(* CODESYS project Fluke.library
   Company: Ziga Javornik
   DefaultNamespace: ZigaLibs.Fluke
   Version: 0.0.1.0
   Placeholder: ZigaLibs.Fluke
   Author: Ziga Javornik
   Title: ZigaLibs.Fluke

Project tree, tasks and I/O mapping:
  libraries: Tc2_Standard, * (Beckhoff Automation GmbH); Tc2_System, * (Beckhoff Automation GmbH); Tc3_Module, * (Beckhoff Automation GmbH); TcUnit, 1.3.1 (www.tcunit.org); ZigaLibs.Core, 0.0.3.7 (Ziga Javornik); ZigaLibs.Logging, 0.0.4.1 (Ziga Javornik); ZigaLibs.TcpIp, 0.0.2.2 (Ziga Javornik)
  GVLs/
  SOURCE/
    Endurance IR Pyrometers/
      DUTs/
        data type ST_EndurancePyrometerCommands
        data type ST_EndurancePyrometerCommParameters
        data type ST_EndurancePyrometerErrorCodes
        data type ST_EndurancePyrometerErrorResponse
      GVLs/
        global variables GVL_Params_EndurancePyrometer
      POUs/
        program EndurancePyrometerConstants [ST]
        function block FB_EndurancePyrometer [ST]: FB_init, CreateSendCommand, ExtractResponse, GetLogPrefix, LogError, LogInfo, LogWarning, RemoveResponsePrefix, RemoveResponseSuffix, ValidateLogger, CommParameters
  TESTS/
    Test suites/
      function block FB_EndurancePyrometer_Tests [ST]: Test00_AttenuationTooHigh_ExpectMaxTemp, Test01_HeaterTemperatureOverrange_ExpectMaxTemp, Test02_HeaterTemperatureUnderrange_ExpectMaxTemp, Test03_InternalTemperatureTooHigh_ExpectMaxTemp, Test04_InternalTemperatureTooLow_ExpectMaxTemp, Test05_SyntaxError_ExpectMaxTemp, Test06_TemperatureOverrange_ExpectMaxTemp, Test07_TemperatureUnderrange_ExpectMinTemp
      function block FB_EndurancePyrometerConstants_Tests [ST]: Test01_ErrorCodesValues
    program PRG_TESTS [ST]
*)

// SOURCE/Endurance IR Pyrometers/DUTs/ST_EndurancePyrometerCommands
TYPE ST_EndurancePyrometerCommands :
STRUCT
	ReadTemperatureCommand 			: STRING := '?T';	// Asks the pyrometer for current temperature
	ReadSensorInternalTemperature	: STRING := '?I';	// Asks for the internal temperature of the sensor
	ReadTargetTemperatureEnergy		: STRING := '?Q';	// Asks for the energy value of the target temperature
	ReadEmissivity					: STRING := '?E';	// Asks for the current emissivity value
	SetEmissivity					: STRING := 'E=';	// Command for setting emissivity, followed value will be set
	SetTemperatuerPhysicalUnit_C	: STRING := 'U=C';	// Sets the physical unit for temperature to °C
	SetTemperatuerPhysicalUnit_F	: STRING := 'U=F';	// Sets the physical unit for temperature to °F
	
	ResponseSuffix			: STRING := '$R$N';	// Response from pyrometer ends with the suffix
	ResponsePrefix			: STRING := '!';	// Response from pyrometer starts with the prefix
	CommandSuffix 			: STRING := '$R';	// Every command needs to end with the suffix
END_STRUCT
END_TYPE

// SOURCE/Endurance IR Pyrometers/DUTs/ST_EndurancePyrometerCommParameters
TYPE ST_EndurancePyrometerCommParameters :
STRUCT
	ReadCycle		: TIME := T#500MS;	// Cyclic reading of certain values is executed within the interval defined by this parameter.
	ReconnectPeriod	: TIME := T#45S;	// Reconnect period for TCP/IP. Don't set too low (30s should be the lowest)
	Ipv4Address		: Tc2_System.T_IPv4Addr := '192.168.42.132';	// IPV4 address of the device.
	Port			: ZigaLibs_TcpIp.T_Port := 6363;	// Port of the device.
END_STRUCT
END_TYPE

// SOURCE/Endurance IR Pyrometers/DUTs/ST_EndurancePyrometerErrorCodes
(*When an error or failure does occur, the temperature display indicates the possible failure area and the output
circuits automatically adjust to the lowest or highest preset level. The following table shows the corresponding
values and the error code transmitted over the digital interface.

Fail safe error codes, from: https://media.fluke.com/048723ef-592e-4cbc-86d4-b4ad00bf9a87_original%20file.pdf

Condition 											2-color 			1-color(wide band)**	1-color*(narrow band)**
Heater temperature over range, >= 80°C (176°F) 		ECHH 				ECHH 					ECHH
Heater temperature under range, <= 50°C (122°F) 	ECUU 				ECUU 					ECUU
Internal temperature over range, >= 85°C (185°F) 	EIHH 				EIHH 					EIHH
Internal temperature under range, <= 0°C (32°F) 	EIUU 				EIUU 					EIUU
Wide band detector failure 							EHHH	 			EHHH 					<temperature>
Narrow band detector failure 						EHHH 				<temperature> 			EHHH
Energy too low 										EUUU 				<temperature> 			<temperature>
Attenuation too high (>95%)*** 						EAAA 				<temperature> 			<temperature>
Attenuation too high >95%
("dirty lens", relay will go to “alarm” state)***	<temperature> 		<temperature> 			<temperature>
2-color temperature under range 					EUUU 				<temperature> 			<temperature>
2-color temperature over range 						EHHH 				<temperature> 			<temperature>
Wide band temperature under range 					<temperature> 		EUUU 					<temperature>
Wide band temperature over range 					<temperature> 		EHHH 					<temperature>
Narrow band temperature under range 				<temperature> 		<temperature> 			EUUU
Narrow band temperature over range 					<temperature> 		<temperature> 			EHHH


* only available via ASCII command
** wide and narrow band stands for the first and the second wavelength in 2-color mode
*** note that the activation levels for these conditions may be set to different values (e.g., "dirty lens" at 95%, EAAA at 98%)
*)
TYPE ST_EndurancePyrometerErrorCodes :
STRUCT
	TemperatureOverrange		: ST_EndurancePyrometerErrorResponse := (Code := 'EHHH', Message := 'Temperature over  range');
	TemperatureUnderrange		: ST_EndurancePyrometerErrorResponse := (Code := 'EUUU', Message := 'Temperature under range');
	InternalTemperatureTooLow	: ST_EndurancePyrometerErrorResponse := (Code := 'EIUU', Message := 'Internal temperature under range, <= 0°C (32°F) ');
	InternalTemperatureTooHigh	: ST_EndurancePyrometerErrorResponse := (Code := 'EIHH', Message := 'Internal temperature over range, >= 85°C (185°F)');
	AttenuationTooHigh			: ST_EndurancePyrometerErrorResponse := (Code := 'EAAA', Message := 'Attenuation too high (>95%)');
	HeaterTemperatureUnderrange	: ST_EndurancePyrometerErrorResponse := (Code := 'ECUU', Message := 'Heater temperature under range, <= 50°C (122°F) ');
	HeaterTemperatureOverrange	: ST_EndurancePyrometerErrorResponse := (Code := 'ECHH', Message := 'Heater temperature over range, >= 80°C (176°F)');
	SyntaxError					: ST_EndurancePyrometerErrorResponse := (Code := '*Syntax Error', Message := 'A value entered in an incorrect format');
END_STRUCT
END_TYPE

// SOURCE/Endurance IR Pyrometers/DUTs/ST_EndurancePyrometerErrorResponse
TYPE ST_EndurancePyrometerErrorResponse :
STRUCT
	Code	: Tc2_System.T_MaxString;
	Message	: STRING;
END_STRUCT
END_TYPE

// SOURCE/Endurance IR Pyrometers/GVLs/GVL_Params_EndurancePyrometer
{attribute 'qualified_only'}
VAR_GLOBAL CONSTANT
	MAX_TEMPERATURE	: REAL := 3000.0;	// Sets the maximum temperature of the pyromerer - should be set accordingly to pyrometer series
	MIN_TEMPERATURE	: REAL := 1000.0;	// Sets the minimum temperatuer of the pyrometer - should be set accordingly to pyrometer series
END_VAR

// SOURCE/Endurance IR Pyrometers/POUs/EndurancePyrometerConstants
PROGRAM EndurancePyrometerConstants
VAR CONSTANT
	ErrorCodes	: ST_EndurancePyrometerErrorCodes;
	Commands	: ST_EndurancePyrometerCommands;	
END_VAR

END_PROGRAM

// SOURCE/Endurance IR Pyrometers/POUs/FB_EndurancePyrometer
FUNCTION_BLOCK FB_EndurancePyrometer EXTENDS ZigaLibs_Core.FB_HasInstanceNameAndPath
VAR_INPUT
	connect		: BOOL;
	readCycle	: TIME;	// Read cycle, should not be set under 300ms, limitation is done within
	ipAddress	: Tc2_System.T_IPv4Addr;
	port		: UINT;	
END_VAR

VAR_OUTPUT
	temperature	: REAL;
	error		: BOOL;
	connected	: BOOL;
	errorCode	: Tc2_System.T_MaxString;
END_VAR

VAR
	_tcpIp			: ZigaLibs_TcpIp.FB_TcpIpCommControl(_logger);
	_reconnectTimer	: Tc2_Standard.TON;
	_readTimer		: Tc2_Standard.TON;
	_readWriteStep	:(READY, SEND_READ_COMMAND, AWAIT_RESPONSE);
	_response		: Tc2_System.T_MaxString;
	_logger			: REFERENCE TO ZigaLibs_Logging.I_Logger;
	_commParameters	: ST_EndurancePyrometerCommParameters;
	_readTemperatureCommand	: STRING;	
	_sb				: ZigaLibs_Core.FB_StringBuilder;
END_VAR

_tcpIp.ReconnectPeriod := T#10S;

_reconnectTimer(
	IN := NOT _reconnectTimer.Q AND _tcpIp.Error, 
	PT := T#30S);

// Communication via TcpIp
IF connect THEN
	IF _reconnectTimer.Q THEN
		_tcpIp.Disconnect();
	ELSIF NOT _tcpIp.IsConnected THEN
		_tcpIp.Connect(ipAddress, port);		
	END_IF
ELSE
	_tcpIp.Disconnect();
END_IF

connected := _tcpIp.IsConnected;
_tcpIp();

IF _tcpIp.IsConnected THEN
	_readTimer(PT := MIN (T#200MS, readCycle));
	
	CASE _readWriteStep OF
		READY:
			_readTimer.IN := TRUE;
			IF _readTimer.Q THEN
				_readTimer.IN := FALSE;
				_readWriteStep := SEND_READ_COMMAND;
			END_IF
		
		SEND_READ_COMMAND:
			_readTemperatureCommand := CreateSendCommand(EndurancePyrometerConstants.Commands.ReadTemperatureCommand);
			IF _tcpIp.Send(_readTemperatureCommand) THEN
				_readWriteStep := AWAIT_RESPONSE;
			END_IF
		
		AWAIT_RESPONSE:
			IF _tcpIp.Receive(_response) THEN
				ExtractResponse('T');
				_readWriteStep := READY;
			END_IF
	END_CASE
ELSE
	// Tcp error - set temperature to max to prevent PID overheating.
	temperature := GVL_Params_EndurancePyrometer.MAX_TEMPERATURE;
END_IF

error := _tcpIp.Error OR error;

METHOD FB_init : BOOL
VAR_INPUT
	bInitRetains : BOOL; // if TRUE, the retain variables are initialized (warm start / cold start)
	bInCopyCode : BOOL;  // if TRUE, the instance afterwards gets moved into the copy code (online change)
	logger	: REFERENCE TO ZigaLibs_Logging.I_Logger;
END_VAR
_logger REF= logger;
END_METHOD

METHOD CreateSendCommand : STRING
VAR_INPUT
	command	: STRING;
END_VAR
CreateSendCommand := Tc2_Standard.CONCAT(command, EndurancePyrometerConstants.Commands.CommandSuffix);
END_METHOD

METHOD INTERNAL ExtractResponse
VAR_INPUT
	sentCommand	: STRING;
END_VAR

VAR
	response			: Tc2_System.T_MaxString;
	responseTmp			: Tc2_System.T_MaxString;
	suffixLength		: INT;

	suffixRemoveAttempt	: DINT;
END_VAR

VAR_INST
	syntaxErrorTrigger	: Tc2_Standard.R_TRIG;
	errorTrigger		: Tc2_Standard.R_TRIG;
	errorClearedTrigge	: Tc2_Standard.F_TRIG;
	sb					: ZigaLibs_Core.FB_StringBuilder;
END_VAR
response := _response;
syntaxErrorTrigger();

// Syntax error - return early
IF Tc2_Standard.FIND(response, EndurancePyrometerConstants.ErrorCodes.SyntaxError.Code) <> 0 THEN
	syntaxErrorTrigger(CLK := TRUE);
	IF syntaxErrorTrigger.Q THEN
		LogError(_sb.Reset()
			.AddString('Syntax error! Sent command is ')
			.AddWithDblQuotationMarks(sentCommand)
			.AddString('.')
			.Create());
	END_IF
	error := TRUE;
	errorCode := 'Syntax error';
	temperature := GVL_Params_EndurancePyrometer.MAX_TEMPERATURE;
	RETURN;
END_IF

syntaxErrorTrigger.CLK := FALSE;

response := RemoveResponsePrefix(sentCommand, response);	
response := RemoveResponseSuffix(response);

error := FALSE;

// Parse response
IF response = EndurancePyrometerConstants.ErrorCodes.TemperatureOverrange.Code THEN
	errorCode := EndurancePyrometerConstants.ErrorCodes.TemperatureOverrange.Message;
	temperature := GVL_Params_EndurancePyrometer.MAX_TEMPERATURE;
ELSIF response = EndurancePyrometerConstants.ErrorCodes.TemperatureUnderrange.Code THEN
	errorCode := EndurancePyrometerConstants.ErrorCodes.TemperatureUnderrange.Message;	
	temperature := GVL_Params_EndurancePyrometer.MIN_TEMPERATURE;	
ELSIF response = EndurancePyrometerConstants.ErrorCodes.InternalTemperatureTooLow.Code THEN
	errorCode := EndurancePyrometerConstants.ErrorCodes.InternalTemperatureTooLow.Message;
	temperature := GVL_Params_EndurancePyrometer.MAX_TEMPERATURE;
	error := TRUE;	
ELSIF response = EndurancePyrometerConstants.ErrorCodes.InternalTemperatureTooHigh.Code THEN
	errorCode := EndurancePyrometerConstants.ErrorCodes.InternalTemperatureTooHigh.Message;
	temperature := GVL_Params_EndurancePyrometer.MAX_TEMPERATURE;
	error := TRUE;	
ELSIF response = EndurancePyrometerConstants.ErrorCodes.AttenuationTooHigh.Code THEN
	errorCode := EndurancePyrometerConstants.ErrorCodes.AttenuationTooHigh.Message;
	temperature := GVL_Params_EndurancePyrometer.MAX_TEMPERATURE;
	error := TRUE;	
ELSIF response = EndurancePyrometerConstants.ErrorCodes.HeaterTemperatureUnderrange.Code THEN
	errorCode := EndurancePyrometerConstants.ErrorCodes.HeaterTemperatureUnderrange.Message;
	temperature := GVL_Params_EndurancePyrometer.MAX_TEMPERATURE;
	error := TRUE;	
ELSIF response = EndurancePyrometerConstants.ErrorCodes.HeaterTemperatureOverrange.Code THEN
	errorCode := EndurancePyrometerConstants.ErrorCodes.HeaterTemperatureOverrange.Message;
	temperature := GVL_Params_EndurancePyrometer.MAX_TEMPERATURE;
	error := TRUE;	
ELSE	
	errorCode := 'No error';
	temperature := STRING_TO_REAL(response);	
END_IF

errorTrigger(CLK := errorCode <> 'No error');
IF errorTrigger.Q THEN
	IF __ISVALIDREF(_logger) THEN
		_logger.LogError(_sb.Reset()
			.AddString(GetLogPrefix())
			.AddString('Pyrometer response indicates error! Error description: ')
			.AddWithDblQuotationMarks(errorCode)
			.AddString('.')
			.Create());
	END_IF	
END_IF

errorClearedTrigge(CLK := errorCode = 'No error');
IF errorClearedTrigge.Q THEN
	IF __ISVALIDREF(_logger) THEN
		_logger.LogInfo(_sb.Reset()
			.AddString(GetLogPrefix())
			.AddString('Previous pyrometer error code is no longer active.')
			.Create());
	END_IF	
END_IF
END_METHOD

METHOD PROTECTED GetLogPrefix : T_MaxString
VAR_INPUT
END_VAR

VAR
	sb	: ZigaLibs_Core.FB_StringBuilder;
END_VAR
GetLogPrefix := sb.AddString(THIS^.InstanceName)
	.AddString(' ')
	.AddWithDblQuotationMarks(ipAddress)
	.AddString(': ')
	.Create();
END_METHOD

METHOD PROTECTED LogError
VAR_INPUT
	message	: Tc2_System.T_MaxString;
END_VAR 
VAR
	sb	: ZigaLibs_Core.FB_StringBuilder;
END_VAR
IF NOT ValidateLogger() THEN
	RETURN;
END_IF

_logger.LogError(
	sb.AddString(GetLogPrefix())
		.AddString(message)
		.Create());
END_METHOD

METHOD PROTECTED LogInfo
VAR_INPUT
	message	: Tc2_System.T_MaxString;
END_VAR 
VAR
	sb	: ZigaLibs_Core.FB_StringBuilder;
END_VAR
IF NOT ValidateLogger() THEN
	RETURN;
END_IF

_logger.LogInfo(
	sb.AddString(GetLogPrefix())
		.AddString(message)
		.Create());
END_METHOD

METHOD PROTECTED LogWarning
VAR_INPUT
	message : Tc2_System.T_MaxString;
END_VAR
VAR
	sb	: ZigaLibs_Core.FB_StringBuilder;
END_VAR
IF NOT ValidateLogger() THEN
	RETURN;
END_IF

_logger.LogWarning(
	sb.AddString(GetLogPrefix())
		.AddString(message)
		.Create());
END_METHOD

// Removes the prefix from the received response and returns the trimmer string
METHOD PROTECTED RemoveResponsePrefix : Tc2_System.T_MaxString
VAR_INPUT
	sentCommand	: Tc2_System.T_MaxString;
	response	: Tc2_System.T_MaxString;
END_VAR
// Remove prefix
RemoveResponsePrefix := Tc2_Standard.DELETE(
	STR := response, 
	LEN := Tc2_Standard.LEN(sentCommand) + LEN(EndurancePyrometerConstants.Commands.ResponsePrefix),
	POS := 1);
END_METHOD

// Removes the suffix from the received response and returns the trimmer string
METHOD PROTECTED RemoveResponseSuffix : T_MaxString
VAR_INPUT
	response	: STRING;
END_VAR
VAR
	suffixPosition	: INT;	
	trimmedResponse		: STRING;
END_VAR

// Remove suffix - sometimes the suffix is sent in multiples (no idea why Fluke does this), remove all occurences!	
suffixPosition := Tc2_Standard.FIND(STR1 := response, STR2 := EndurancePyrometerConstants.Commands.ResponseSuffix);
trimmedResponse := response;
IF suffixPosition <> 0 THEN
	response := Tc2_Standard.LEFT(STR := trimmedResponse, SIZE := suffixPosition - 1);		
END_IF

RemoveResponseSuffix := trimmedResponse;
END_METHOD

METHOD PROTECTED ValidateLogger : BOOL
VAR_INPUT
END_VAR
ValidateLogger := __ISVALIDREF(_logger);
END_METHOD

// Gets or sets communication parameters of the device.
PROPERTY PUBLIC CommParameters : REFERENCE TO ST_EndurancePyrometerCommParameters
GET
CommParameters REF= _commParameters;
END_GET
SET
_commParameters := CommParameters;
END_SET
END_PROPERTY

END_FUNCTION_BLOCK

// TESTS/Test suites/FB_EndurancePyrometer_Tests
// Subject under test
FUNCTION_BLOCK INTERNAL FB_EndurancePyrometer_Tests EXTENDS FB_TestSuite

// Create instance variables that will be accesible for all tests
VAR
END_VAR

// Call your test methods here
Test00_AttenuationTooHigh_ExpectMaxTemp();
Test01_HeaterTemperatureOverrange_ExpectMaxTemp();
Test02_HeaterTemperatureUnderrange_ExpectMaxTemp();
Test03_InternalTemperatureTooHigh_ExpectMaxTemp();
Test04_InternalTemperatureTooLow_ExpectMaxTemp();
Test05_SyntaxError_ExpectMaxTemp();
Test06_TemperatureOverrange_ExpectMaxTemp();
Test07_TemperatureUnderrange_ExpectMinTemp();

METHOD PRIVATE Test00_AttenuationTooHigh_ExpectMaxTemp

(* Instanced variables are VERY useful for writing tests since tests are run in paralel (by default).
By instantiating local variables that are not placed on the same stack as method (values are retained between calls)
you make sure that the SUT is not changed by some other test. *)
VAR_INST
	
END_VAR

// Place temporary variables here
VAR
	pyrometer	: FB_EndurancePyrometer(0);
END_VAR
// The name of the test, is the same as method name!
// Use this for paralel unit tests
// TcUnit.TEST('TestXX_Template');

// Use this for running tests in sequence
IF TcUnit.TEST_ORDERED('Test00_AttenuationTooHigh_ExpectMaxTemp') THEN
	
	TcUnit.WRITE_PROTECTED_STRING(
		ADR(pyrometer._response), 
		CONCAT('!T', EndurancePyrometerConstants.ErrorCodes.AttenuationTooHigh.Code));
		
	pyrometer.ExtractResponse('T');
	AssertEquals_REAL(
		Actual := pyrometer.temperature,
		Expected := GVL_Params_EndurancePyrometer.MAX_TEMPERATURE,
		Delta := 0.1,
		Message := '');
		
	AssertTrue(Condition := pyrometer.error, Message := 'Attenuation too high should trigger an error');
	TcUnit.TEST_FINISHED();	
END_IF
END_METHOD

METHOD PRIVATE Test01_HeaterTemperatureOverrange_ExpectMaxTemp

(* Instanced variables are VERY useful for writing tests since tests are run in paralel (by default).
By instantiating local variables that are not placed on the same stack as method (values are retained between calls)
you make sure that the SUT is not changed by some other test. *)
VAR_INST
	
END_VAR

// Place temporary variables here
VAR
	pyrometer	: FB_EndurancePyrometer(0);
END_VAR
// The name of the test, is the same as method name!
// Use this for paralel unit tests
// TcUnit.TEST('TestXX_Template');

// Use this for running tests in sequence
IF TcUnit.TEST_ORDERED('Test01_HeaterTemperatureOverrange_ExpectMaxTemp') THEN
	
	TcUnit.WRITE_PROTECTED_STRING(
		ADR(pyrometer._response), 
		CONCAT('!T', EndurancePyrometerConstants.ErrorCodes.HeaterTemperatureOverrange.Code));
		
	pyrometer.ExtractResponse('T');
	AssertEquals_REAL(
		Actual := pyrometer.temperature,
		Expected := GVL_Params_EndurancePyrometer.MAX_TEMPERATURE,
		Delta := 0.1,
		Message := '');

	AssertTrue(Condition := pyrometer.error, Message := 'Heater temperature overrange should trigger an error');
	TcUnit.TEST_FINISHED();	
END_IF
END_METHOD

METHOD PRIVATE Test02_HeaterTemperatureUnderrange_ExpectMaxTemp

(* Instanced variables are VERY useful for writing tests since tests are run in paralel (by default).
By instantiating local variables that are not placed on the same stack as method (values are retained between calls)
you make sure that the SUT is not changed by some other test. *)
VAR_INST
	
END_VAR

// Place temporary variables here
VAR
	pyrometer	: FB_EndurancePyrometer(0);
END_VAR
// The name of the test, is the same as method name!
// Use this for paralel unit tests
// TcUnit.TEST('TestXX_Template');

// Use this for running tests in sequence
IF TcUnit.TEST_ORDERED('Test02_HeaterTemperatureUnderrange_ExpectMaxTemp') THEN
	
	TcUnit.WRITE_PROTECTED_STRING(
		ADR(pyrometer._response), 
		CONCAT('!T', EndurancePyrometerConstants.ErrorCodes.HeaterTemperatureUnderrange.Code));
		
	pyrometer.ExtractResponse('T');
	AssertEquals_REAL(
		Actual := pyrometer.temperature,
		Expected := GVL_Params_EndurancePyrometer.MAX_TEMPERATURE,
		Delta := 0.1,
		Message := '');
		
	AssertTrue(Condition := pyrometer.error, Message := ' Heater temperature underrange should trigger an error');		
	TcUnit.TEST_FINISHED();	
END_IF
END_METHOD

METHOD PRIVATE Test03_InternalTemperatureTooHigh_ExpectMaxTemp

(* Instanced variables are VERY useful for writing tests since tests are run in paralel (by default).
By instantiating local variables that are not placed on the same stack as method (values are retained between calls)
you make sure that the SUT is not changed by some other test. *)
VAR_INST
	
END_VAR

// Place temporary variables here
VAR
	pyrometer	: FB_EndurancePyrometer(0);
END_VAR
// The name of the test, is the same as method name!
// Use this for paralel unit tests
// TcUnit.TEST('TestXX_Template');

// Use this for running tests in sequence
IF TcUnit.TEST_ORDERED('Test03_InternalTemperatureTooHigh_ExpectMaxTemp') THEN
	
	TcUnit.WRITE_PROTECTED_STRING(
		ADR(pyrometer._response), 
		CONCAT('!T', EndurancePyrometerConstants.ErrorCodes.InternalTemperatureTooHigh.Code));
		
	pyrometer.ExtractResponse('T');
	AssertEquals_REAL(
		Actual := pyrometer.temperature,
		Expected := GVL_Params_EndurancePyrometer.MAX_TEMPERATURE,
		Delta := 0.1,
		Message := '');
		
	AssertTrue(Condition := pyrometer.error, Message := 'Internal temperature too high should trigger an error');	
	TcUnit.TEST_FINISHED();	
END_IF
END_METHOD

METHOD PRIVATE Test04_InternalTemperatureTooLow_ExpectMaxTemp

(* Instanced variables are VERY useful for writing tests since tests are run in paralel (by default).
By instantiating local variables that are not placed on the same stack as method (values are retained between calls)
you make sure that the SUT is not changed by some other test. *)
VAR_INST
	
END_VAR

// Place temporary variables here
VAR
	pyrometer	: FB_EndurancePyrometer(0);
END_VAR
// The name of the test, is the same as method name!
// Use this for paralel unit tests
// TcUnit.TEST('TestXX_Template');

// Use this for running tests in sequence
IF TcUnit.TEST_ORDERED('Test04_InternalTemperatureTooLow_ExpectMaxTemp') THEN
	
	TcUnit.WRITE_PROTECTED_STRING(
		ADR(pyrometer._response), 
		CONCAT('!T', EndurancePyrometerConstants.ErrorCodes.InternalTemperatureTooLow.Code));
		
	pyrometer.ExtractResponse('T');
	AssertEquals_REAL(
		Actual := pyrometer.temperature,
		Expected := GVL_Params_EndurancePyrometer.MAX_TEMPERATURE,
		Delta := 0.1,
		Message := '');
		
	AssertTrue(Condition := pyrometer.error, Message := 'Internal tempereature too low should trigger an error');	
	TcUnit.TEST_FINISHED();	
END_IF
END_METHOD

METHOD PRIVATE Test05_SyntaxError_ExpectMaxTemp

(* Instanced variables are VERY useful for writing tests since tests are run in paralel (by default).
By instantiating local variables that are not placed on the same stack as method (values are retained between calls)
you make sure that the SUT is not changed by some other test. *)
VAR_INST
	
END_VAR

// Place temporary variables here
VAR
	pyrometer	: FB_EndurancePyrometer(0);
END_VAR
// The name of the test, is the same as method name!
// Use this for paralel unit tests
// TcUnit.TEST('TestXX_Template');

// Use this for running tests in sequence
IF TcUnit.TEST_ORDERED('Test05_SyntaxError_ExpectMaxTemp') THEN
	
	TcUnit.WRITE_PROTECTED_STRING(
		ADR(pyrometer._response), 
		CONCAT('!T', EndurancePyrometerConstants.ErrorCodes.SyntaxError.Code));
		
	pyrometer.ExtractResponse('T');
	AssertEquals_REAL(
		Actual := pyrometer.temperature,
		Expected := GVL_Params_EndurancePyrometer.MAX_TEMPERATURE,
		Delta := 0.1,
		Message := '');
		
	AssertTrue(Condition := pyrometer.error, Message := 'Syntax error should trigger an error');	
	TcUnit.TEST_FINISHED();	
END_IF
END_METHOD

METHOD PRIVATE Test06_TemperatureOverrange_ExpectMaxTemp

(* Instanced variables are VERY useful for writing tests since tests are run in paralel (by default).
By instantiating local variables that are not placed on the same stack as method (values are retained between calls)
you make sure that the SUT is not changed by some other test. *)
VAR_INST
	
END_VAR

// Place temporary variables here
VAR
	pyrometer	: FB_EndurancePyrometer(0);
END_VAR
// The name of the test, is the same as method name!
// Use this for paralel unit tests
// TcUnit.TEST('TestXX_Template');

// Use this for running tests in sequence
IF TcUnit.TEST_ORDERED('Test06_TemperatureOverrange_ExpectMaxTemp') THEN
	
	TcUnit.WRITE_PROTECTED_STRING(
		ADR(pyrometer._response), 
		CONCAT('!T', EndurancePyrometerConstants.ErrorCodes.TemperatureOverrange.Code));
		
	pyrometer.ExtractResponse('T');
	AssertEquals_REAL(
		Actual := pyrometer.temperature,
		Expected := GVL_Params_EndurancePyrometer.MAX_TEMPERATURE,
		Delta := 0.1,
		Message := '');
		
	AssertFalse(Condition := pyrometer.error, Message := 'Temperature overrange should not trigger an error');	
	TcUnit.TEST_FINISHED();	
END_IF
END_METHOD

METHOD PRIVATE Test07_TemperatureUnderrange_ExpectMinTemp

(* Instanced variables are VERY useful for writing tests since tests are run in paralel (by default).
By instantiating local variables that are not placed on the same stack as method (values are retained between calls)
you make sure that the SUT is not changed by some other test. *)
VAR_INST
	
END_VAR

// Place temporary variables here
VAR
	pyrometer	: FB_EndurancePyrometer(0);
END_VAR
// The name of the test, is the same as method name!
// Use this for paralel unit tests
// TcUnit.TEST('TestXX_Template');

// Use this for running tests in sequence
IF TcUnit.TEST_ORDERED('Test07_TemperatureUnderrange_ExpectMinTemp') THEN
	
	TcUnit.WRITE_PROTECTED_STRING(
		ADR(pyrometer._response), 
		CONCAT('!T', EndurancePyrometerConstants.ErrorCodes.TemperatureUnderrange.Code));
		
	pyrometer.ExtractResponse('T');
	AssertEquals_REAL(
		Actual := pyrometer.temperature,
		Expected := GVL_Params_EndurancePyrometer.MIN_TEMPERATURE,
		Delta := 0.1,
		Message := '');
	
	AssertFalse(Condition := pyrometer.error, Message := 'Temperature underrange should not trigger an error');	
	TcUnit.TEST_FINISHED();	
END_IF
END_METHOD

END_FUNCTION_BLOCK

// TESTS/Test suites/FB_EndurancePyrometerConstants_Tests
FUNCTION_BLOCK INTERNAL FB_EndurancePyrometerConstants_Tests EXTENDS FB_TestSuite
VAR_INPUT
END_VAR
VAR_OUTPUT
END_VAR
VAR
END_VAR

Test01_ErrorCodesValues();

METHOD PRIVATE Test01_ErrorCodesValues
(*
Fail safe error codes, from: https://media.fluke.com/048723ef-592e-4cbc-86d4-b4ad00bf9a87_original%20file.pdf

Condition 											2-color 			1-color(wide band)**	1-color*(narrow band)**
Heater temperature over range, >= 80°C (176°F) 		ECHH 				ECHH 					ECHH
Heater temperature under range, <= 50°C (122°F) 	ECUU 				ECUU 					ECUU
Internal temperature over range, >= 85°C (185°F) 	EIHH 				EIHH 					EIHH
Internal temperature under range, <= 0°C (32°F) 	EIUU 				EIUU 					EIUU
Wide band detector failure 							EHHH	 			EHHH 					<temperature>
Narrow band detector failure 						EHHH 				<temperature> 			EHHH
Energy too low 										EUUU 				<temperature> 			<temperature>
Attenuation too high (>95%)*** 						EAAA 				<temperature> 			<temperature>
[Attenuation too high >95%
("dirty lens", relay will go to “alarm” state)***]	<temperature> 		<temperature> 			<temperature>
2-color temperature under range 					EUUU 				<temperature> 			<temperature>
2-color temperature over range 						EHHH 				<temperature> 			<temperature>
Wide band temperature under range 					<temperature> 		EUUU 					<temperature>
Wide band temperature over range 					<temperature> 		EHHH 					<temperature>
Narrow band temperature under range 				<temperature> 		<temperature> 			EUUU
Narrow band temperature over range 					<temperature> 		<temperature> 			EHHH


* only available via ASCII command
** wide and narrow band stands for the first and the second wavelength in 2-color mode
*** note that the activation levels for these conditions may be set to different values (e.g., "dirty lens" at 95%, EAAA at 98%)
*)
IF TcUnit.TEST_ORDERED('Test01_ErrorCodesValues') THEN
	
	AssertEquals_STRING(
		Actual := EndurancePyrometerConstants.ErrorCodes.TemperatureOverrange.Code,
		Expected := 'EHHH',
		Message := 'Temperature overrange code is incorrect');
		
	AssertEquals_STRING(
		Actual := EndurancePyrometerConstants.ErrorCodes.TemperatureUnderrange.Code,
		Expected := 'EUUU',
		Message := 'Temperature underrange code is incorrect');
		
	AssertEquals_STRING(
		Actual := EndurancePyrometerConstants.ErrorCodes.InternalTemperatureTooLow.Code,
		Expected := 'EIUU',
		Message := 'Internal temperature too low code is incorrect');
		
	AssertEquals_STRING(
		Actual := EndurancePyrometerConstants.ErrorCodes.InternalTemperatureTooHigh.Code,
		Expected := 'EIHH',
		Message := 'Internal temperature too high code is incorrect');
		
	AssertEquals_STRING(
		Actual := EndurancePyrometerConstants.ErrorCodes.AttenuationTooHigh.Code,
		Expected := 'EAAA',
		Message := 'Attenutation too high code is incorrect');
		
	AssertEquals_STRING(
		Actual := EndurancePyrometerConstants.ErrorCodes.HeaterTemperatureUnderrange.Code,
		Expected := 'ECUU',
		Message := 'Heater temperature underrange code is incorrect');	
		
	AssertEquals_STRING(
		Actual := EndurancePyrometerConstants.ErrorCodes.HeaterTemperatureOverrange.Code,
		Expected := 'ECHH',
		Message := 'Heater temperature overrange code is incorrect');	
		
	AssertEquals_STRING(
		Actual := EndurancePyrometerConstants.ErrorCodes.SyntaxError.Code,
		Expected := '*Syntax Error',
		Message := 'Syntax error code is incorrect');	
		
	TcUnit.TEST_FINISHED();
END_IF
END_METHOD

END_FUNCTION_BLOCK

// TESTS/PRG_TESTS
PROGRAM INTERNAL PRG_TESTS

(* Instantiate test suites here. Naming convention for tests should be a suffix with _Tests.
Good practice for creating test methods is to end them with _test as well. *)

VAR
	EndurancePyrometer_Tests			: FB_EndurancePyrometer_Tests;
	EndurancePyrometerConstants_Tests	: FB_EndurancePyrometerConstants_Tests;
END_VAR

// Run tests in parallel
//TcUnit.RUN();

// Run tests in sequence, one after the other.
TcUnit.RUN_IN_SEQUENCE();

END_PROGRAM
